SUBAPPLICATION mapping_Uebung_028 (* Subapplication Type *)
  (* Standard: 61499-2 *)
  (* Version 1.0, 2023-10-23, franz *)
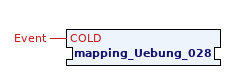
  EVENT_INPUT
    COLD;
  END_EVENT
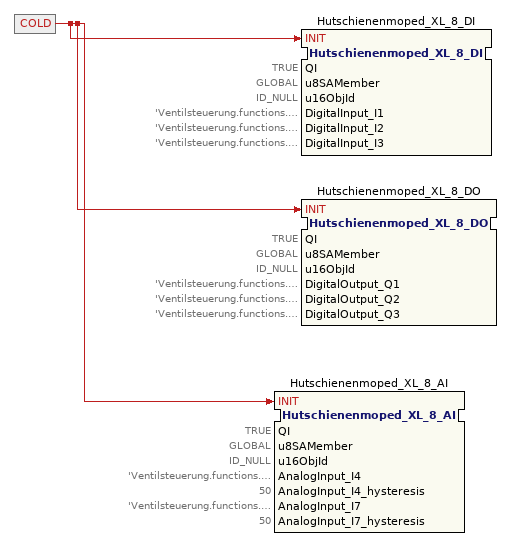
  FBS
    Hutschienenmoped_XL_8_DO : Hutschienenmoped_XL_8_DO(QI := TRUE, u8SAMember := GLOBAL, u16ObjId := ID_NULL, DigitalOutput_Q1 := 'Ventilsteuerung.functions.DigitalOutput_Q1', DigitalOutput_Q2 := 'Ventilsteuerung.functions.DigitalOutput_Q2', DigitalOutput_Q3 := 'Ventilsteuerung.functions.DigitalOutput_Q3');
    Hutschienenmoped_XL_8_DI : Hutschienenmoped_XL_8_DI(QI := TRUE, u8SAMember := GLOBAL, u16ObjId := ID_NULL, DigitalInput_I1 := 'Ventilsteuerung.functions.DigitalInput_I1', DigitalInput_I2 := 'Ventilsteuerung.functions.DigitalInput_I2', DigitalInput_I3 := 'Ventilsteuerung.functions.DigitalInput_I3');
    Hutschienenmoped_XL_8_AI : Hutschienenmoped_XL_8_AI(QI := TRUE, u8SAMember := GLOBAL, u16ObjId := ID_NULL, AnalogInput_I4 := 'Ventilsteuerung.functions.AnalogInput_I4', AnalogInput_I4_hysteresis := 50, AnalogInput_I7 := 'Ventilsteuerung.functions.AnalogInput_I7', AnalogInput_I7_hysteresis := 50);
  END_FBS
  EVENT_CONNECTIONS
    COLD TO Hutschienenmoped_XL_8_DI.INIT;
    COLD TO Hutschienenmoped_XL_8_DO.INIT;
    COLD TO Hutschienenmoped_XL_8_AI.INIT;
  END_CONNECTIONS
END_SUBAPPLICATION
